{attribute 'GeneratedUsingTerminal: EP2339-0021-0016'}
{attribute addProperty BoxType "EP2339-0021-0016"}
{attribute addProperty Id "AoeNetIdAT %I*.TcoAmsNetId0StateAT %I*UINT2"}
{attribute addProperty CRC "131947802"}
{attribute addProperty Size "2"}
TYPE InfoData_07DD5D1A :
STRUCT
	{attribute addProperty Name "AoeNetId"}
	AoeNetId AT %I* : .TcoAmsNetId;
	{attribute addProperty Name "State"}
	State AT %I* : UINT;
END_STRUCT
END_TYPE

(* stored: Version 1.2.0.0, ProductVersion 3.1.4024.9
   DUT InfoData_07DD5D1A: Id {fdb34a3e-53cf-4778-a1f6-f8efa393962f} *)
